Staubli VAL3: start.pgx

program start()
begin
  while true
    sTest="0123456789"
    sTest1=left(sTest[0],1)
  endWhile
end
